// TIA Portal V16 export
// export: Created 2024-06-24T15:42:27.4565019Z, ExportSetting WithDefaults, DisplayName Totally Integrated Automation Portal, DisplayVersion V16, DisplayName TIA Portal Version Control Interface, DisplayVersion V16, DisplayName TIA Portal Openness, DisplayVersion V16, DisplayName STEP 7 Professional, DisplayVersion V16, DisplayName STEP 7 Safety, DisplayVersion V16, DisplayName WinCC Advanced, DisplayVersion V16
ORGANIZATION_BLOCK "OB_Line_Init"   // OB125, LAD, ProgramCycle
TITLE = "Main Program Sweep (Cycle)"
{ S7_Optimized_Access := 'TRUE' }
VERSION : 0.1
// stored: AutoNumber true, IsIECCheckEnabled false, SetENOAutomatically false
   VAR_INPUT
      Initial_Call : Bool;   // Initial call of this OB
      Remanence : Bool;   // =True, if remanent data are available
   END_VAR
   VAR_TEMP   // added for the SCL form of the ladder/FBD networks
      _w1 : Bool;
   END_VAR
BEGIN

REGION Network 1
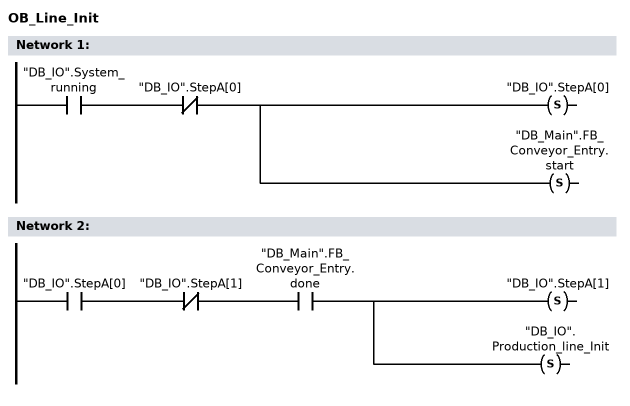
   RUNG wire#powerrail
      Contact( "DB_IO".System_running )
      I_Contact( "DB_IO".StepA[0] )
      wire#w1
      S_Coil( "DB_IO".StepA[0] )
   END_RUNG
   RUNG wire#w1
      S_Coil( "DB_Main".FB_Conveyor_Entry.start )
   END_RUNG
   // the same network as SCL:
   #_w1 := "DB_IO".System_running AND NOT "DB_IO".StepA[0];
   IF #_w1 THEN
       "DB_IO".StepA[0] := TRUE;
       "DB_Main".FB_Conveyor_Entry.start := TRUE;
   END_IF;
END_REGION

REGION Network 2
   RUNG wire#powerrail
      Contact( "DB_IO".StepA[0] )
      I_Contact( "DB_IO".StepA[1] )
      Contact( "DB_Main".FB_Conveyor_Entry.done )
      wire#w1
      S_Coil( "DB_IO".StepA[1] )
   END_RUNG
   RUNG wire#w1
      S_Coil( "DB_IO".Production_line_Init )
   END_RUNG
   // the same network as SCL:
   #_w1 := "DB_IO".StepA[0] AND NOT "DB_IO".StepA[1] AND "DB_Main".FB_Conveyor_Entry.done;
   IF #_w1 THEN
       "DB_IO".StepA[1] := TRUE;
       "DB_IO".Production_line_Init := TRUE;
   END_IF;
END_REGION
END_ORGANIZATION_BLOCK
